PROGRAM P2_05_SP_Process_Ctrl
VAR
	tonProcessTime					:FB_TONP;
	tonActiveProcessTime			:FB_TONP;
	tProcessTime					:TIME;
END_VAR

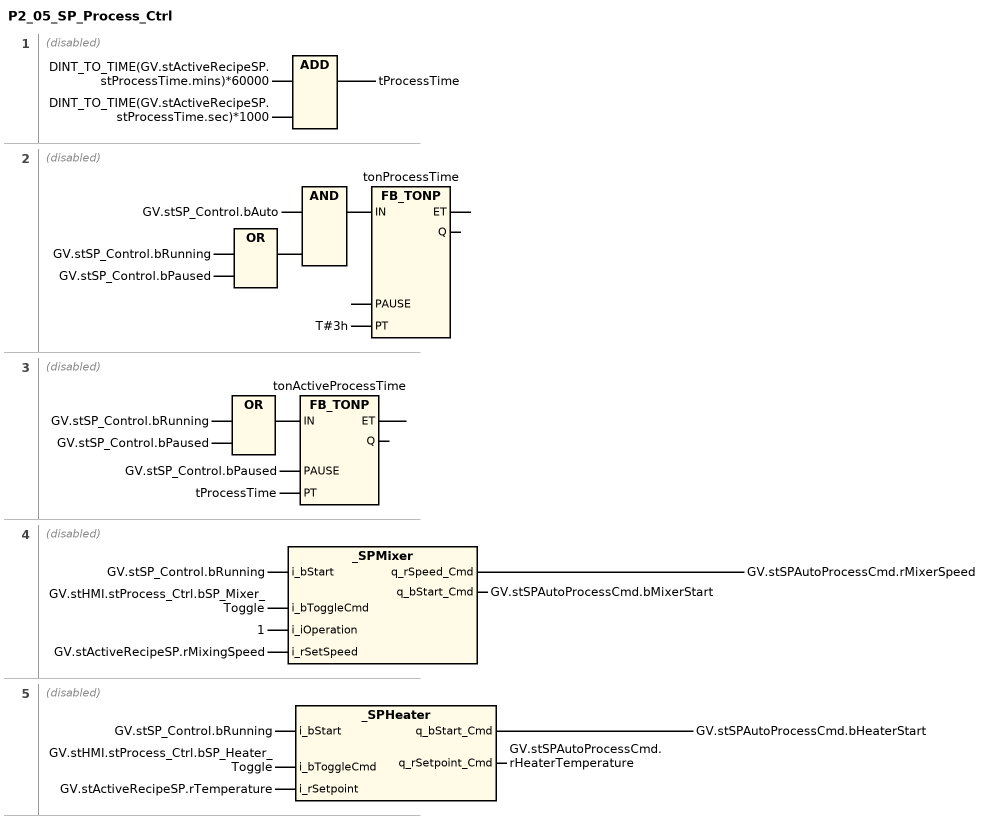
// NETWORK 1 (disabled)
// tProcessTime := (DINT_TO_TIME(GV.stActiveRecipeSP.stProcessTime.mins)*60000) + (DINT_TO_TIME(GV.stActiveRecipeSP.stProcessTime.sec)*1000);

// NETWORK 2 (disabled)
// tonProcessTime(IN := GV.stSP_Control.bAuto AND (GV.stSP_Control.bRunning OR GV.stSP_Control.bPaused), PT := T#3h); // FB_TONP

// NETWORK 3 (disabled)
// tonActiveProcessTime(
//     IN := GV.stSP_Control.bRunning OR GV.stSP_Control.bPaused,
//     PAUSE := GV.stSP_Control.bPaused,
//     PT := tProcessTime); // FB_TONP

// NETWORK 4 (disabled)
// _SPMixer(i_bStart := GV.stSP_Control.bRunning, i_bToggleCmd := GV.stHMI.stProcess_Ctrl.bSP_Mixer_Toggle, i_iOperation := 1, i_rSetSpeed := GV.stActiveRecipeSP.rMixingSpeed, q_bStart_Cmd => GV.stSPAutoProcessCmd.bMixerStart);
// GV.stSPAutoProcessCmd.rMixerSpeed := _SPMixer.q_rSpeed_Cmd;

// NETWORK 5 (disabled)
// _SPHeater(i_bStart := GV.stSP_Control.bRunning, i_bToggleCmd := GV.stHMI.stProcess_Ctrl.bSP_Heater_Toggle, i_rSetpoint := GV.stActiveRecipeSP.rTemperature, q_rSetpoint_Cmd => GV.stSPAutoProcessCmd.rHeaterTemperature);
// GV.stSPAutoProcessCmd.bHeaterStart := _SPHeater.q_bStart_Cmd;

END_PROGRAM

(* stored: Version 1.1.0.1, ProductVersion 3.1.4026.13
   POU P2_05_SP_Process_Ctrl: Id {3f7774ba-2466-4ea7-835f-cc60c4fb7178}, SpecialFunc None *)
